PROGRAM Main_T10ms
VAR

END_VAR

Simulation();

Monitoring();

END_PROGRAM

(* stored: Version 1.1.0.1, ProductVersion 3.1.4024.12
   POU Main_T10ms: Id {6779098e-183c-40bc-9866-f079e3b788e4}, SpecialFunc None *)
